// TIA Portal V16 export
// export: Created 2021-08-30T11:09:37.5525994Z, ExportSetting WithDefaults, DisplayName Totally Integrated Automation Portal, DisplayVersion V16 Update 3, DisplayName TIA Portal Version Control Interface, DisplayVersion V16 Update 2, DisplayName TIA Portal Openness, DisplayVersion V16 Update 3, DisplayName TIA Portal Teamcenter Gateway, DisplayVersion V16, DisplayName STEP 7 Professional, DisplayVersion V16 Update 3, DisplayName STEP 7 Safety, DisplayVersion V16, DisplayName WinCC Advanced, DisplayVersion V16 Update 3
TYPE "ET_HW_AQ"
// stored: IsFailsafeCompliant false
   STRUCT
      HW_AQ : Array[0.."ET_AQ"] of Int;
   END_STRUCT;
END_TYPE
